# EPICS substitutions: iocs/aerotechIOC/iocBoot/iocAerotech/Ensemble.substitutions
file "$(MOTOR)/db/asyn_motor.db"
{
pattern
{P,          N,     M,      DTYP,         PORT,   ADDR,  DESC,          EGU,  DIR,  VELO,  VBAS,  ACCL,  BDST,  BVEL,  BACC,  MRES,   PREC,  DHLM,  DLLM,          INIT}
{aerotech:,  1,  "m$(N)",  "asynMotor",  AeroE1,    0,  "motor $(N)",  mm,   Pos,  .1,     0,    .2,    0,     1,     .2,    1.25E-5,   7,     0,      0,  "SCURVE 100"}
}
